Staubli VAL3: Rob6x.dtx

mdesc mNomSpeed = {accel=50, vel=20, decel=50, tmax=1000, leave=10, reach=10, blend=off}
tool tGripper3Sucks = {z=200, rx=-180, fatherId=flange[0], ioLink=valve1}
pointRx pPointHome = {x=200, fatherId=world[0]}
bool bExit
sio siTcpServer = {link=Socket\Server}
tool tCurrentTool = {fatherId=flange[0], ioLink=valve1}
bool AlignMode
pointRx pPointsTable{}
num LastErrorCode
num GeneralStatus
num CurLimitsTable{}
pointRx pTargetPoint = {fatherId=world[0]}
jointRx jTargetJoint
num FrameReceiveOK
num FrameReceiveNOK
frame fCurrentFrame = {fatherId=world[0]}
bool AsyncMode
sio siTcpClient = {link=Socket\Client}
bool ExecuteMotion
bool CartesianMode
jointRx jHome = {j3=90}
bool MotionTaskMutex
num NbCharReceived
dio diVacuum = {link=fIn0}
dio doPump = {link=fOut0}
dio difIn1 = {link=fIn1}
dio diusrIn0 = {link=usrIn0}
dio diusrIn1 = {link=usrIn1}
dio doValve2 = {link=valve2}
num currentToolType
tool tGripper4Sucks = {z=200, rx=-180, fatherId=flange[0], ioLink=valve1}
tool tPICC_ISO = {x=160.4, z=200, rx=-180, fatherId=flange[0], ioLink=valve1}
tool tPICC_NFC = {x=137.46, z=200, rx=-180, fatherId=flange[0], ioLink=valve1}
tool tPICC_EMV = {x=127.7, z=200, rx=-180, fatherId=flange[0], ioLink=valve1}
jointRx jUser = {j3=90, j5=90}
bool MoveRunning
bool bStartRecording
bool bOverload
string sPath
sio siSerial1 = {link=Serial\1}
num NbBufSerial
num BufferSerial[64]
bool ModeSerial
num COEFF_ACCEL
